// TIA Portal project "PLC_Project" (V16)

(* hardware
DEVICE "S7-1200 station_1"  S7-1200 Station
   slot 0: "Rack_0"  S7-1200 Rack  Rack  V1.0
   slot 1: "PLC_1"  CPU 1212C AC/DC/Rly  6ES7 212-1BE40-0XB0  V4.2
   slot 2: "AI 4x13BIT/AQ 2x14BIT_1"  6ES7 234-4HE32-0XB0  V2.1
*)

// ===== PLC "PLC_1"  CPU 1212C AC/DC/Rly =====

VAR_GLOBAL   // PLC tag table "Default tag table"
   "Level Tank 1" AT %IW64 : Int;
   "Level Tank 2" AT %IW66 : Int;
   "StartPump1" AT %I0.0 : Bool;
   "Stop1" AT %I0.1 : Bool;
   "StartPump2" AT %I0.2 : Bool;
   "Stop2" AT %I0.3 : Bool;
   "Level Tank 3" AT %IW96 : Int;
   "Level Tank 4" AT %IW98 : Int;
   "Pump1" AT %Q0.0 : Bool;
   "Pump2" AT %Q0.1 : Bool;
   "Tag_1" AT %QW96 : Int;
   "FV2 Write" AT %QW98 : Int;
   "Level Tank 1 Memory" AT %MD50 : Real;
   "Level Tank 2 Memory" AT %MD58 : Real;
   "FV1 Wirite" AT %MD20 : Real;
   "FV1 Real" AT %MD24 : Real;
   "FV2 Memory" AT %MD28 : Real;
   "FV2 Real" AT %MD32 : Real;
   "Clock_Byte" AT %MB0 : Byte;
   "Clock_10Hz" AT %M0.0 : Bool;
   "Clock_5Hz" AT %M0.1 : Bool;
   "Clock_2.5Hz" AT %M0.2 : Bool;
   "Clock_2Hz" AT %M0.3 : Bool;
   "Clock_1.25Hz" AT %M0.4 : Bool;
   "Clock_1Hz" AT %M0.5 : Bool;
   "Clock_0.625Hz" AT %M0.6 : Bool;
   "Clock_0.5Hz" AT %M0.7 : Bool;
   "Level Tank 3 Memory" AT %MD66 : Real;
   "Level Tank 4 Memory" AT %MD74 : Real;
END_VAR

DATA_BLOCK "Data_PID"   // DB3
{ S7_Optimized_Access := 'FALSE' }
VERSION : 0.1
   VAR
      "PV Tank1" : Real;
      "SP Tank2" : Real;
      "MV Tank1" : Real := 0.0;
      "PV Tank2" : Real := 0.0;
      "MV Tank2" : Real := 0.0;
      "PV Tank3" : Real := -0.003616898;
      "SP Tank4" : Real := 0.0;
      "MV Tank3" : Real := 0.004340277;
      "PV Tank4" : Real := 0.0;
      "MV Tank4" : Real := 0.006926359;
      "SP Tank2 d" : Word;
      "SP Tank4 d" : Word;
      "PV Tank1 d" : Word;
      "PV Tank2 d" : Word;
      "PV Tank3 d" : Word;
      "PV Tank4 d" : Word;
   END_VAR
BEGIN
END_DATA_BLOCK

FUNCTION "Process" : Void   // FC1, LAD
{ S7_Optimized_Access := 'TRUE' }
VERSION : 0.1
BEGIN

REGION Network 1
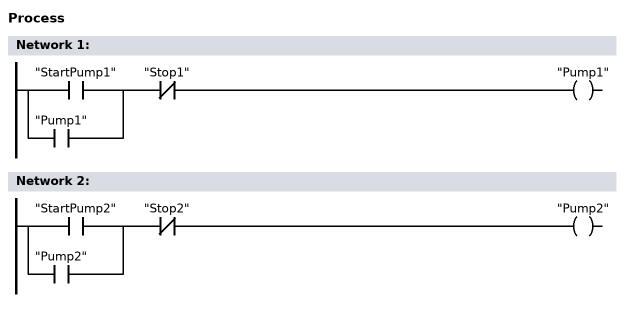
   RUNG wire#powerrail
      Contact( "StartPump1" )
      wire#w1
      I_Contact( "Stop1" )
      Coil( "Pump1" )
   END_RUNG
   RUNG wire#powerrail
      Contact( "Pump1" )
   END_RUNG wire#w1
   // the same network as SCL:
   "Pump1" := ("StartPump1" OR "Pump1") AND NOT "Stop1";
END_REGION

REGION Network 2
   RUNG wire#powerrail
      Contact( "StartPump2" )
      wire#w1
      I_Contact( "Stop2" )
      Coil( "Pump2" )
   END_RUNG
   RUNG wire#powerrail
      Contact( "Pump2" )
   END_RUNG wire#w1
   // the same network as SCL:
   "Pump2" := ("StartPump2" OR "Pump2") AND NOT "Stop2";
END_REGION
END_FUNCTION

FUNCTION "Scale" : Void   // FC2, LAD
{ S7_Optimized_Access := 'TRUE' }
VERSION : 0.1
BEGIN

REGION Network 1: Set point
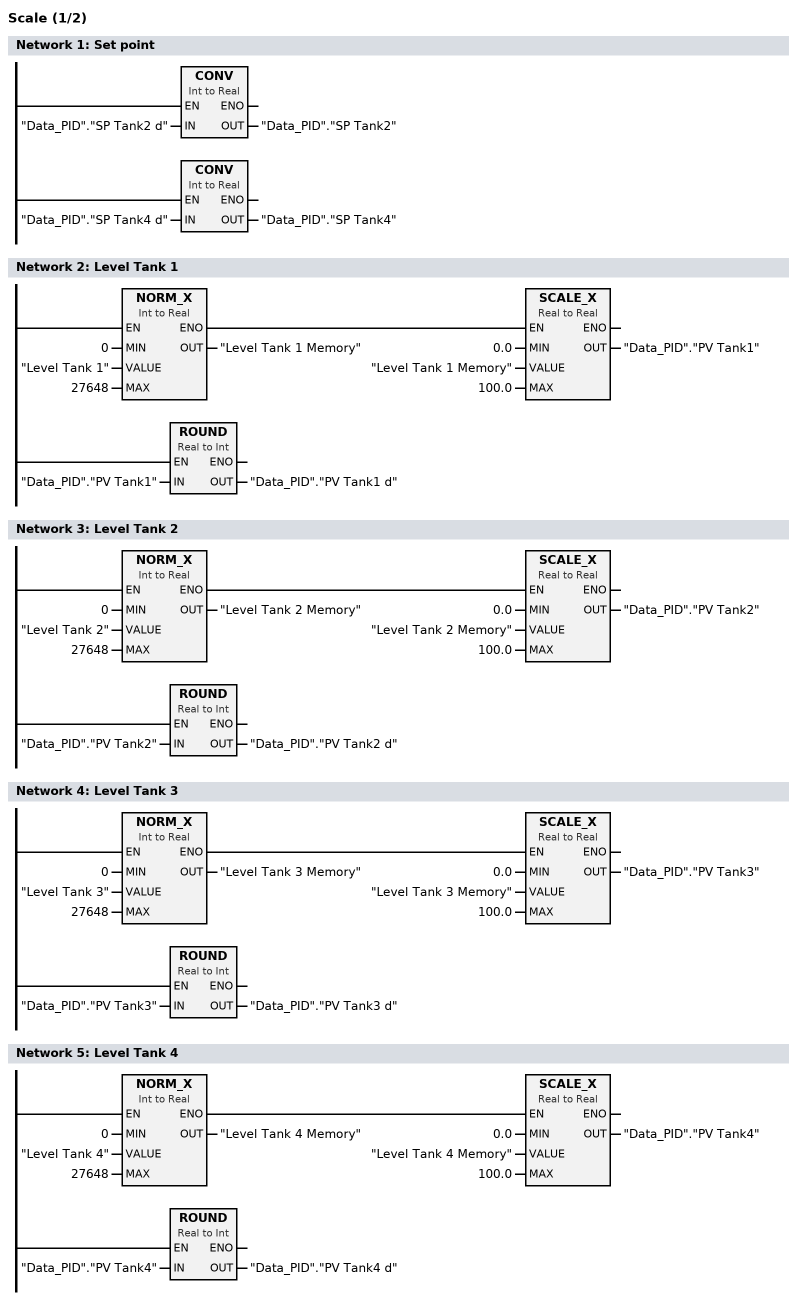
   RUNG wire#powerrail
      { S7_Templates := "[SrcType := Int, DestType := Real]" } Convert(in := "Data_PID"."SP Tank2 d", out => "Data_PID"."SP Tank2")
   END_RUNG
   RUNG wire#powerrail
      { S7_Templates := "[SrcType := Int, DestType := Real]" } Convert(in := "Data_PID"."SP Tank4 d", out => "Data_PID"."SP Tank4")
   END_RUNG
   // the same network as SCL:
   "Data_PID"."SP Tank2" := INT_TO_REAL("Data_PID"."SP Tank2 d");
   "Data_PID"."SP Tank4" := INT_TO_REAL("Data_PID"."SP Tank4 d");
END_REGION

REGION Network 2: Level Tank 1
   RUNG wire#powerrail
      { S7_Templates := "[SrcType := Int, DestType := Real]" } Normalize(min := 0, value := "Level Tank 1", max := 27648, out => "Level Tank 1 Memory")
      { S7_Templates := "[SrcType := Real, DestType := Real]" } Scale(min := 0.0, value := "Level Tank 1 Memory", max := 100.0, out => "Data_PID"."PV Tank1")
   END_RUNG
   RUNG wire#powerrail
      { S7_Templates := "[SrcType := Real, DestType := Int]" } Round(in := "Data_PID"."PV Tank1", out => "Data_PID"."PV Tank1 d")
   END_RUNG
   // the same network as SCL:
   "Level Tank 1 Memory" := NORM_X(MIN := 0, VALUE := "Level Tank 1", MAX := 27648);
   "Data_PID"."PV Tank1" := SCALE_X(MIN := 0.0, VALUE := "Level Tank 1 Memory", MAX := 100.0);
   "Data_PID"."PV Tank1 d" := ROUND("Data_PID"."PV Tank1");
END_REGION

REGION Network 3: Level Tank 2
   RUNG wire#powerrail
      { S7_Templates := "[SrcType := Int, DestType := Real]" } Normalize(min := 0, value := "Level Tank 2", max := 27648, out => "Level Tank 2 Memory")
      { S7_Templates := "[SrcType := Real, DestType := Real]" } Scale(min := 0.0, value := "Level Tank 2 Memory", max := 100.0, out => "Data_PID"."PV Tank2")
   END_RUNG
   RUNG wire#powerrail
      { S7_Templates := "[SrcType := Real, DestType := Int]" } Round(in := "Data_PID"."PV Tank2", out => "Data_PID"."PV Tank2 d")
   END_RUNG
   // the same network as SCL:
   "Level Tank 2 Memory" := NORM_X(MIN := 0, VALUE := "Level Tank 2", MAX := 27648);
   "Data_PID"."PV Tank2" := SCALE_X(MIN := 0.0, VALUE := "Level Tank 2 Memory", MAX := 100.0);
   "Data_PID"."PV Tank2 d" := ROUND("Data_PID"."PV Tank2");
END_REGION

REGION Network 4: Level Tank 3
   RUNG wire#powerrail
      { S7_Templates := "[SrcType := Int, DestType := Real]" } Normalize(min := 0, value := "Level Tank 3", max := 27648, out => "Level Tank 3 Memory")
      { S7_Templates := "[SrcType := Real, DestType := Real]" } Scale(min := 0.0, value := "Level Tank 3 Memory", max := 100.0, out => "Data_PID"."PV Tank3")
   END_RUNG
   RUNG wire#powerrail
      { S7_Templates := "[SrcType := Real, DestType := Int]" } Round(in := "Data_PID"."PV Tank3", out => "Data_PID"."PV Tank3 d")
   END_RUNG
   // the same network as SCL:
   "Level Tank 3 Memory" := NORM_X(MIN := 0, VALUE := "Level Tank 3", MAX := 27648);
   "Data_PID"."PV Tank3" := SCALE_X(MIN := 0.0, VALUE := "Level Tank 3 Memory", MAX := 100.0);
   "Data_PID"."PV Tank3 d" := ROUND("Data_PID"."PV Tank3");
END_REGION

REGION Network 5: Level Tank 4
   RUNG wire#powerrail
      { S7_Templates := "[SrcType := Int, DestType := Real]" } Normalize(min := 0, value := "Level Tank 4", max := 27648, out => "Level Tank 4 Memory")
      { S7_Templates := "[SrcType := Real, DestType := Real]" } Scale(min := 0.0, value := "Level Tank 4 Memory", max := 100.0, out => "Data_PID"."PV Tank4")
   END_RUNG
   RUNG wire#powerrail
      { S7_Templates := "[SrcType := Real, DestType := Int]" } Round(in := "Data_PID"."PV Tank4", out => "Data_PID"."PV Tank4 d")
   END_RUNG
   // the same network as SCL:
   "Level Tank 4 Memory" := NORM_X(MIN := 0, VALUE := "Level Tank 4", MAX := 27648);
   "Data_PID"."PV Tank4" := SCALE_X(MIN := 0.0, VALUE := "Level Tank 4 Memory", MAX := 100.0);
   "Data_PID"."PV Tank4 d" := ROUND("Data_PID"."PV Tank4");
END_REGION

REGION Network 6: % Vavlve1
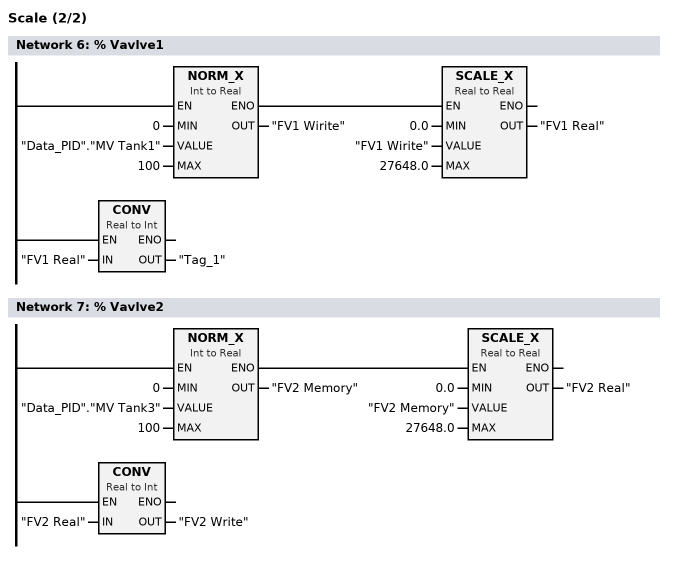
   RUNG wire#powerrail
      { S7_Templates := "[SrcType := Int, DestType := Real]" } Normalize(min := 0, value := "Data_PID"."MV Tank1", max := 100, out => "FV1 Wirite")
      { S7_Templates := "[SrcType := Real, DestType := Real]" } Scale(min := 0.0, value := "FV1 Wirite", max := 27648.0, out => "FV1 Real")
   END_RUNG
   RUNG wire#powerrail
      { S7_Templates := "[SrcType := Real, DestType := Int]" } Convert(in := "FV1 Real", out => "Tag_1")
   END_RUNG
   // the same network as SCL:
   "FV1 Wirite" := NORM_X(MIN := 0, VALUE := "Data_PID"."MV Tank1", MAX := 100);
   "FV1 Real" := SCALE_X(MIN := 0.0, VALUE := "FV1 Wirite", MAX := 27648.0);
   "Tag_1" := REAL_TO_INT("FV1 Real");
END_REGION

REGION Network 7: % Vavlve2
   RUNG wire#powerrail
      { S7_Templates := "[SrcType := Int, DestType := Real]" } Normalize(min := 0, value := "Data_PID"."MV Tank3", max := 100, out => "FV2 Memory")
      { S7_Templates := "[SrcType := Real, DestType := Real]" } Scale(min := 0.0, value := "FV2 Memory", max := 27648.0, out => "FV2 Real")
   END_RUNG
   RUNG wire#powerrail
      { S7_Templates := "[SrcType := Real, DestType := Int]" } Convert(in := "FV2 Real", out => "FV2 Write")
   END_RUNG
   // the same network as SCL:
   "FV2 Memory" := NORM_X(MIN := 0, VALUE := "Data_PID"."MV Tank3", MAX := 100);
   "FV2 Real" := SCALE_X(MIN := 0.0, VALUE := "FV2 Memory", MAX := 27648.0);
   "FV2 Write" := REAL_TO_INT("FV2 Real");
END_REGION
END_FUNCTION

ORGANIZATION_BLOCK "Main"   // OB1, LAD, ProgramCycle
TITLE = "Main Program Sweep (Cycle)"
{ S7_Optimized_Access := 'TRUE' }
VERSION : 0.1
   VAR_INPUT
      Initial_Call : Bool;   // Initial call of this OB
      Remanence : Bool;   // =True, if remanent data are available
   END_VAR
BEGIN

REGION Network 1
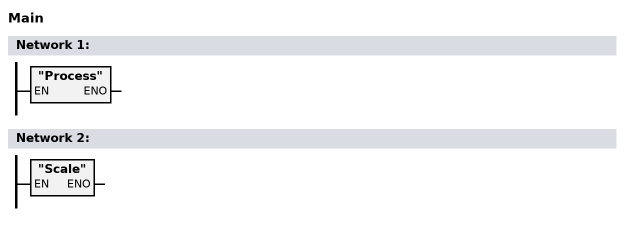
   RUNG wire#powerrail
      "Process"()
   END_RUNG
   // the same network as SCL:
   "Process"();
END_REGION

REGION Network 2
   RUNG wire#powerrail
      "Scale"()
   END_RUNG
   // the same network as SCL:
   "Scale"();
END_REGION
END_ORGANIZATION_BLOCK

ORGANIZATION_BLOCK "Cyclic interrupt (PID)"   // OB30, LAD, CyclicInterrupt
{ S7_Optimized_Access := 'TRUE' }
VERSION : 0.1
   VAR_INPUT
      Initial_Call : Bool;   // Initial call of this OB
      Event_Count : Int;   // Events discarded
   END_VAR
BEGIN

REGION Network 1: Process 1
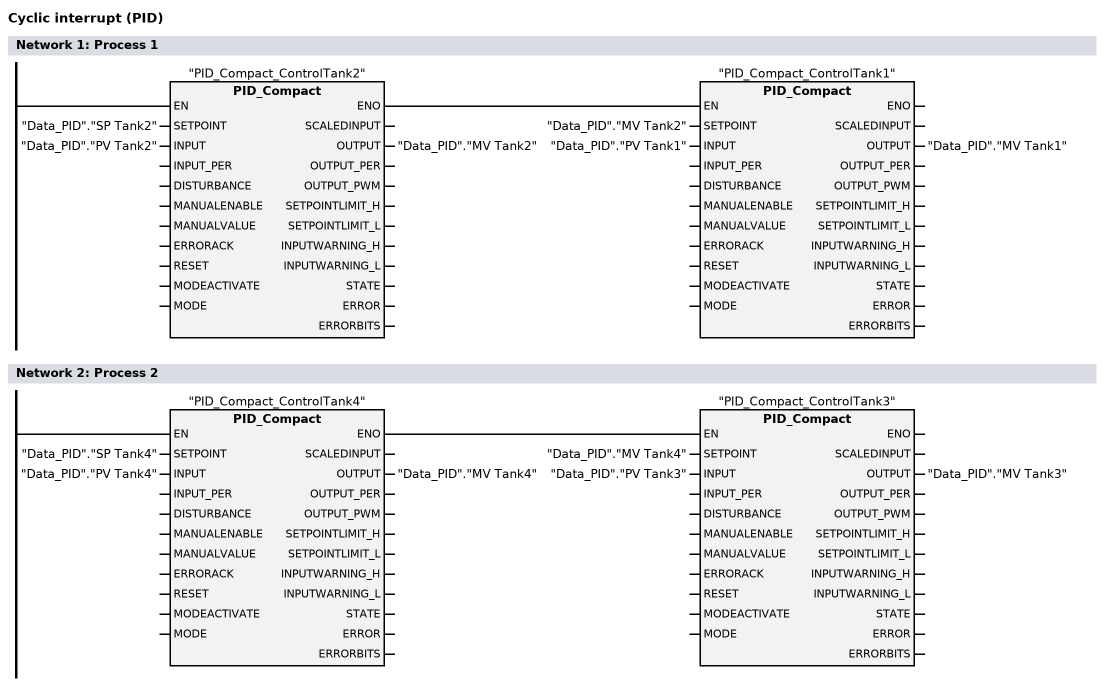
   // ENO of a box is taken as its EN; it also drops when the box reports an error
   "PID_Compact_ControlTank2"(Setpoint := "Data_PID"."SP Tank2",   // PID_Compact
                           Input := "Data_PID"."PV Tank2",
                           Output => "Data_PID"."MV Tank2");
   "PID_Compact_ControlTank1"(Setpoint := "Data_PID"."MV Tank2",   // PID_Compact
                           Input := "Data_PID"."PV Tank1",
                           Output => "Data_PID"."MV Tank1");
END_REGION

REGION Network 2: Process 2
   // ENO of a box is taken as its EN; it also drops when the box reports an error
   "PID_Compact_ControlTank4"(Setpoint := "Data_PID"."SP Tank4",   // PID_Compact
                           Input := "Data_PID"."PV Tank4",
                           Output => "Data_PID"."MV Tank4");
   "PID_Compact_ControlTank3"(Setpoint := "Data_PID"."MV Tank4",   // PID_Compact
                           Input := "Data_PID"."PV Tank3",
                           Output => "Data_PID"."MV Tank3");
END_REGION
END_ORGANIZATION_BLOCK